(* IEC 61131-3 sources: OMBSON/src/Ar/OMBSON, 3 files *)

(* ---- Types.typ ---- *)
(*
 * File: OMBSON.fun
 * Copyright (c) 2023 Loupe
 * https://loupe.team
 *
 * This file is part of OMBSON, licensed under the MIT License.
 *)

TYPE

END_TYPE

(* ---- OMBSON.fun ---- *)
(*
 * File: OMBSON.fun
 * Copyright (c) 2023 Loupe
 * https://loupe.team
 *
 * This file is part of OMBSON, licensed under the MIT License.
 *)

FUNCTION json2bson : UDINT (*Return is the BSON size*) (*$GROUP=User,$CAT=User,$GROUPICON=User.png,$CATICON=User.png*)
	VAR_INPUT
		Bin : UDINT; (*BSON output*)
		Str : UDINT; (*JSON to convert*)
		BufferSize : UDINT; (*Size of Buffer for BSON output*)
	END_VAR
END_FUNCTION

(* ---- Constants.var ---- *)
(*
 * File: Constants.var
 * Copyright (c) 2023 Loupe
 * https://loupe.team
 *
 * This file is part of OMBSON, licensed under the MIT License.
 *)

VAR CONSTANT

END_VAR
